% RSLogix 500 project P1_RIZVI_M.RSS, saved by version 8.10.00.18 %
PROJECT "UNTITLED"    % processor: Bul.1763 MicroLogix 1100 Series B %

PROGRAM FILES
  LAD 2 "MAIN"  3 rungs
  LAD 3 "DIGITAL IO"  5 rungs
  LAD 4 "CONTROLS"  3 rungs

DATA FILES
  O0 OUTPUT  5 elements
  I1 INPUT  7 elements
  S2 STATUS  66 elements
  B3 BINARY  5 elements
  T4 TIMER  1 elements
  C5 COUNTER  1 elements
  R6 CONTROL  1 elements
  N7 INTEGER  1 elements
  F8 FLOAT  1 elements

LADDER 2 "MAIN"
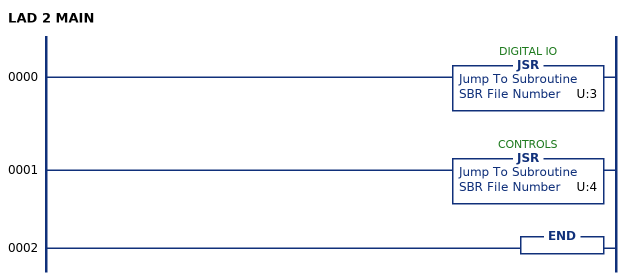
% Rung: 0 %
SOR JSR U:3 EOR
%   U:3  "DIGITAL IO" %
% Rung: 1 %
SOR JSR U:4 EOR
%   U:4  "CONTROLS" %
% Rung: 2 %
SOR END EOR

LADDER 3 "DIGITAL IO"
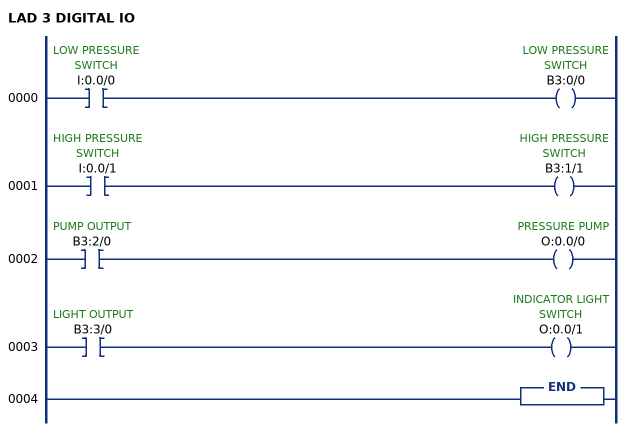
% Rung: 0 %
SOR XIC I:0.0/0 OTE B3:0/0 EOR
%   I:0.0/0  "LOW PRESSURE SWITCH" %
%   B3:0/0  "LOW PRESSURE SWITCH" %
% Rung: 1 %
SOR XIC I:0.0/1 OTE B3:1/1 EOR
%   I:0.0/1  "HIGH PRESSURE SWITCH" %
%   B3:1/1  "HIGH PRESSURE SWITCH" %
% Rung: 2 %
SOR XIC B3:2/0 OTE O:0.0/0 EOR
%   B3:2/0  "PUMP OUTPUT" %
%   O:0.0/0  "PRESSURE PUMP" %
% Rung: 3 %
SOR XIC B3:3/0 OTE O:0.0/1 EOR
%   B3:3/0  "LIGHT OUTPUT" %
%   O:0.0/1  "INDICATOR LIGHT SWITCH" %
% Rung: 4 %
SOR END EOR

LADDER 4 "CONTROLS"
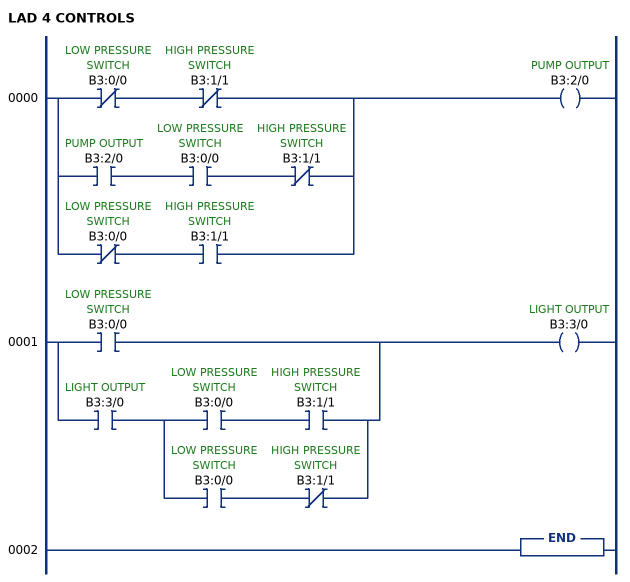
% Rung: 0 %
SOR BST BST XIO B3:0/0 XIO B3:1/1 NXB XIC B3:2/0 XIC B3:0/0 XIO B3:1/1 BND NXB XIO B3:0/0 XIC B3:1/1 BND OTE B3:2/0 EOR
%   B3:0/0  "LOW PRESSURE SWITCH" %
%   B3:1/1  "HIGH PRESSURE SWITCH" %
%   B3:2/0  "PUMP OUTPUT" %
% Rung: 1 %
SOR BST XIC B3:0/0 NXB XIC B3:3/0 BST XIC B3:0/0 XIC B3:1/1 NXB XIC B3:0/0 XIO B3:1/1 BND BND OTE B3:3/0 EOR
%   B3:0/0  "LOW PRESSURE SWITCH" %
%   B3:3/0  "LIGHT OUTPUT" %
%   B3:1/1  "HIGH PRESSURE SWITCH" %
% Rung: 2 %
SOR END EOR

OTHER DOCUMENTED ADDRESSES
  B3:0  "LOW PRESSURE SWITCH"
  B3:0/1  "ONE SHOT"
  B3:1  "HIGH PRESSURE SWITCH"
  B3:2  "PRESSURE PUMP OUTPUT"
  B3:2/1  "PUMP OUTPUT"
  B3:3  "INDICATOR LIGHT OUTPUT"
  B3:4  "One shot"

DATA TABLE (non-zero values as saved)
DATA B3
% B3:0 % 0X0001 0X0000 0X0001 0X0001 0X0000
